TYPE "multicontrolAI_highLevelObjectReady"
TITLE = {"version":"v1.0","author":"cyanezf","family":"core/controller/interroll/multicontrolAI","status":"current","deprecatedBy": null,"dependencies":[]}

//(*--
//# Documentation
//## Log
//| version | date | author | description |
//|:-------:|:----:|:------:|:------------|
//| v1.0 | 2022-10-12 | cyanezf | First version |
//
//## Description
//Multicontrol AI - high-level object ready
//--*)

   STRUCT
      nr : USInt;   // Motor number
      hloReady : Bool;   // 1=High-level object ready (Multicontrol AI)
      ready : Bool;   // 1=This motor is ready
   END_STRUCT;

END_TYPE

